FUNCTION_BLOCK AE_DELAY (* Delayed event propagation (AE Adapter) *)
  (* Standard: 61499-2; Description: Copyright (c) 2026 HR Agrartechnik GmbH This program and the accompanying materials are made available under the terms of the Eclipse Public License 2.0 which is available at https://www.eclipse.org/legal/epl-2.0/ SPDX-License-Identifier: EPL-2.0 *)
  (* Version 1.0, 2026-02-01, Franz Höpfinger, HR Agrartechnik GmbH, Wrapper for E_DELAY using AE adapters *)
  (* Version 1.1, 2026-09-17, Franz Höpfinger, HR Agrartechnik GmbH, Bugfix (Franz: 'DT ... muesste dann auch einen ATM als TIME Eingang bekommen'): Klartext-InputVar DT:TIME (nie ueber INIT initialisiert) durch ATM-Socket ersetzt, sauber initialisierbar ueber initval_ATM+INIT/INITO an der Instanziierungsstelle. Toter, unverdrahteter EventInput REQ (Rest einer Kopiervorlage) mit entfernt. *)
  (* Version 1.2, 2026-09-17, Franz Höpfinger, HR Agrartechnik GmbH, Bugfix (4diac IDE Validation: 'Name: DT is a reserved keyword' - DT ist Abkuerzung fuer DATE_AND_TIME, IEC 61131-3-Keyword): Socket DT in PT (Preset Time, Standardname wie bei TON/TOF) umbenannt. *)
  PACKAGE adapter::events::unidirectional::timers;
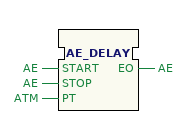
  SOCKETS
    START : adapter::types::unidirectional::AE; (* Start delay *)
    STOP : adapter::types::unidirectional::AE; (* Stop delay *)
    PT : adapter::types::unidirectional::ATM; (* Preset Time / Delay time (ATM statt Klartext-InputVar, sauber initialisierbar ueber initval_ATM) *)
  END_SOCKETS
  PLUGS
    EO : adapter::types::unidirectional::AE; (* Delayed event *)
  END_PLUGS
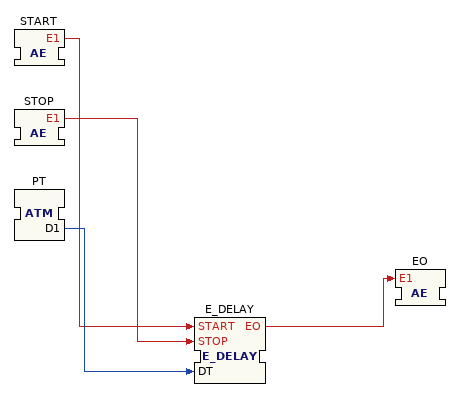
  FBS
    E_DELAY : iec61499::events::E_DELAY;
  END_FBS
  EVENT_CONNECTIONS
    START.E1 TO E_DELAY.START;
    STOP.E1 TO E_DELAY.STOP;
    E_DELAY.EO TO EO.E1;
  END_CONNECTIONS
  DATA_CONNECTIONS
    PT.D1 TO E_DELAY.DT;
  END_CONNECTIONS
END_FUNCTION_BLOCK
